{attribute 'GeneratedUsingTerminal: AES-D-BC-ECAT Gen2-0001'}
{attribute addProperty BoxType "AES-D-BC-ECAT Gen2-0001"}
{attribute addProperty Id "digital_Data_OAT %Q*ARRAY[0..31] OF USINT32"}
{attribute addProperty CRC "2024821696"}
{attribute addProperty Size "32"}
TYPE Outputs_FC2FACAD EXTENDS TcoIo.OutputBase_10CEE7DE :
STRUCT
	{attribute addProperty Name "digital_Data_O"}
	digital_Data_O AT %Q* : ARRAY[0..31] OF USINT;
END_STRUCT
END_TYPE

(* stored: Version 1.2.0.0
   DUT Outputs_FC2FACAD: Id {81d01f40-6449-4ff6-9639-1aa3d36582a8} *)
